// TIA Portal V16 export
// export: Created 2021-05-18T09:41:03.9474871Z, ExportSetting WithDefaults, DisplayName Totally Integrated Automation Portal, DisplayVersion V16 Update 3, DisplayName TIA Portal Version Control Interface, DisplayVersion V16 Update 2, DisplayName TIA Portal Openness, DisplayVersion V16 Update 3, DisplayName STEP 7 Professional, DisplayVersion V16 Update 3, DisplayName STEP 7 Safety, DisplayVersion V16, DisplayName WinCC Professional, DisplayVersion V16 Update 3
DATA_BLOCK "DB02001_St_InstAnalogRead"   // DB2001
TITLE = Static DB — Inst - Analog Instrument Read, Scale and Monitor
{ S7_Optimized_Access := 'TRUE' }
AUTHOR : M_Gledhill
FAMILY : Instrumentation
NAME : St_InstAnalogRead
VERSION : 0.1
// PRACTICAL SERIES AUTOMATION LIBRARY (PAL)   —   COPYRIGHT 2020 – M. GLEDHILL (MIT LICENCE)
//                   ———— ◆ ————
//  FOR DETAILED DOCUMENTATION — SELECT THE BLOCK IN THE PROJECT TREE AND PRESS SHIFT + F1
//  FULL ONLINE DOCUMENTATION IS AVAILABLE AT: https://practicalseries.com/2001-pal/index.html
// stored: AutoNumber false, DBAccessibleFromOPCUA true, IsOnlyStoredInLoadMemory false, IsRetainMemResEnabled false, IsWriteProtectedInAS false, MemoryReserve 100
   VAR
      _DB_Header { ExternalAccessible := 'False'; ExternalVisible := 'False'; ExternalWritable := 'False'} : Array[0..79] of Bool;   // STANDARD ANALOG INSTRUMENT READ
      __________0000_0 { ExternalAccessible := 'False'; ExternalVisible := 'False'; ExternalWritable := 'False'} : Bool := false;
      __________0000_1 { ExternalAccessible := 'False'; ExternalVisible := 'False'; ExternalWritable := 'False'} : Bool := false;   // ▀▀▀▀ DB CURRENT REVISION
      revInfo { ExternalWritable := 'False'; S7_SetPoint := 'True'} : "UT01000_St_SysRevision";
      __________0010_0 { ExternalAccessible := 'False'; ExternalVisible := 'False'; ExternalWritable := 'False'} : Bool := false;
      __________0010_1 { ExternalAccessible := 'False'; ExternalVisible := 'False'; ExternalWritable := 'False'} : Bool := false;   // ▀▀▀▀ ANALOG INSTRUMENTS
      FIC101 { ExternalWritable := 'False'; S7_SetPoint := 'True'} : "UT02001_St_InstAnalogRead";   // Filter 1 outlet flow
   END_VAR
BEGIN
   // _DB_Header[0] : ▀▀▀▀▀▀▀▀▀▀▀▀▀▀▀▀▀▀▀▀▀▀▀▀▀▀▀▀▀▀▀▀▀▀▀▀▀▀▀▀▀▀▀▀
   // _DB_Header[2] : TITLE: STANDARD ANALOG INSTRUMENT READ (SCALE & ALARM MONITORING)
   // _DB_Header[4] : ▄▄▄▄▄▄▄▄▄▄▄▄▄▄▄▄▄▄▄▄▄▄▄▄▄▄▄▄▄▄▄▄▄▄▄▄▄▄▄▄▄▄▄▄
   // _DB_Header[5] : TYPE: STATIC
   // _DB_Header[6] : ▀▀▀▀▀▀▀▀▀▀▀▀▀▀▀▀▀▀▀▀▀▀▀▀▀▀▀▀▀▀▀▀▀▀▀▀▀▀▀▀▀▀▀▀
   // _DB_Header[8] : This is the static data block associated with the standard analog instrument read
   // _DB_Header[9] : block:
   // _DB_Header[10] : FC02001_StdInstAnalogRead
   // _DB_Header[12] : The static data holds the threshold values for any configured alarms and warnings,
   // _DB_Header[13] : activation delays, scaled and raw value ranges and various configuration options.
   // _DB_Header[15] : Each instrument is given the user data type:
   // _DB_Header[16] : UT02001_St_InstAnalogRead
   // _DB_Header[17] : This holds the full set of static configuration data for the instrument.
   // _DB_Header[19] : ━━━ ⬙⬙⬙⬙⬙⬙ ━━━
   // _DB_Header[21] : ▄▄▄▄▄▄▄▄▄▄▄▄▄▄▄▄▄▄▄▄▄▄▄▄▄▄▄▄▄▄▄▄▄▄▄▄▄▄▄▄▄▄▄▄
   // _DB_Header[22] : MODIFICATION HISTORY
   // _DB_Header[24] : This is a summary of the recent software modifications made to this block (most recent at top)
   // _DB_Header[26] : ―――――――――――――――――――――――――――――――――――――――――――
   // _DB_Header[27] : DATE REVISION MASTER BRANCH DEV
   // _DB_Header[28] : (nnn.amm) COMMIT TAG (Base ---> Merge) BRANCH Author
   // _DB_Header[29] : ———————————————————————————————————————————
   // _DB_Header[30] : 2021.05.18 000.101 D0006B-000.101 D0006 N/A D0006B M. Gledhill
   // _DB_Header[31] : FC02001 Migration to VCS
   // _DB_Header[32] : ———————————————————————————————————————————
   // _DB_Header[33] : Where: nnn = Major revision
   // _DB_Header[34] : a = Type (1-7 Development, 8 Proving, 9 Qualification, 0 Release)
   // _DB_Header[35] : mm = Minor revision (must be 00 if a = 0)
   // _DB_Header[36] : Block properties version number should be set to nn.a (only one decimal place)
   // _DB_Header[38] : ██████████████ █ █ █ █ END █ █ █ █ ██████████████
   revInfo.REV_BLOCK := 'DB02001';
   revInfo.REV_NUMBER := '000.101';
   revInfo.REV_DATE := '2021-05-18';
   revInfo.REV_AUTHOR := 'M. Gledhill';
   FIC101.CONFIG_ALM_H_ENABLE := true;
   FIC101.CONFIG_ALM_L_ENABLE := true;
   FIC101.CONFIG_WRN_H_ENABLE := true;
   FIC101.CONFIG_WRN_L_ENABLE := true;
   FIC101.CONFIG_FP_DISABLE := false;
   FIC101.CONFIG_SIM_DISABLE := false;
   FIC101.CONFIG_RL_ENABLE := false;
   FIC101.RANGE_RAW_MAX := 27648;
   FIC101.RANGE_SCALE_MIN := 0.0;
   FIC101.RANGE_SCALE_MAX := 1000.0;
   FIC101.RANGE_OOR_PERCENT := 2.5;
   FIC101.INFO_TAG := 'FIC101';
   FIC101.INFO_UNITS := 'l/s';
   FIC101.SP_ALM_H_VAL := 750.0;
   FIC101.SP_ALM_L_VAL := 250.0;
   FIC101.SP_WRN_H_VAL := 625.0;
   FIC101.SP_WRN_L_VAL := 375.0;
   FIC101.SP_ALM_H_HYST_VAL := 62.5;
   FIC101.SP_ALM_L_HYST_VAL := 62.0;
   FIC101.SP_WRN_H_HYST_VAL := 61.5;
   FIC101.SP_WRN_L_HYST_VAL := 61.0;
   FIC101.TIME_ALM_H_ON_DEL := 10.0;
   FIC101.TIME_ALM_L_ON_DEL := 11.0;
   FIC101.TIME_WRN_H_ON_DEL := 12.0;
   FIC101.TIME_WRN_L_ON_DEL := 13.0;
   FIC101.TIME_ALM_H_OFF_DEL := 15.0;
   FIC101.TIME_ALM_L_OFF_DEL := 16.0;
   FIC101.TIME_WRN_H_OFF_DEL := 17.0;
   FIC101.TIME_WRN_L_OFF_DEL := 18.0;
END_DATA_BLOCK
